// Mitsubishi GX Works2 project: For_daiverter2   PLC: FX3U/FX3UC

PROGRAM MAIN
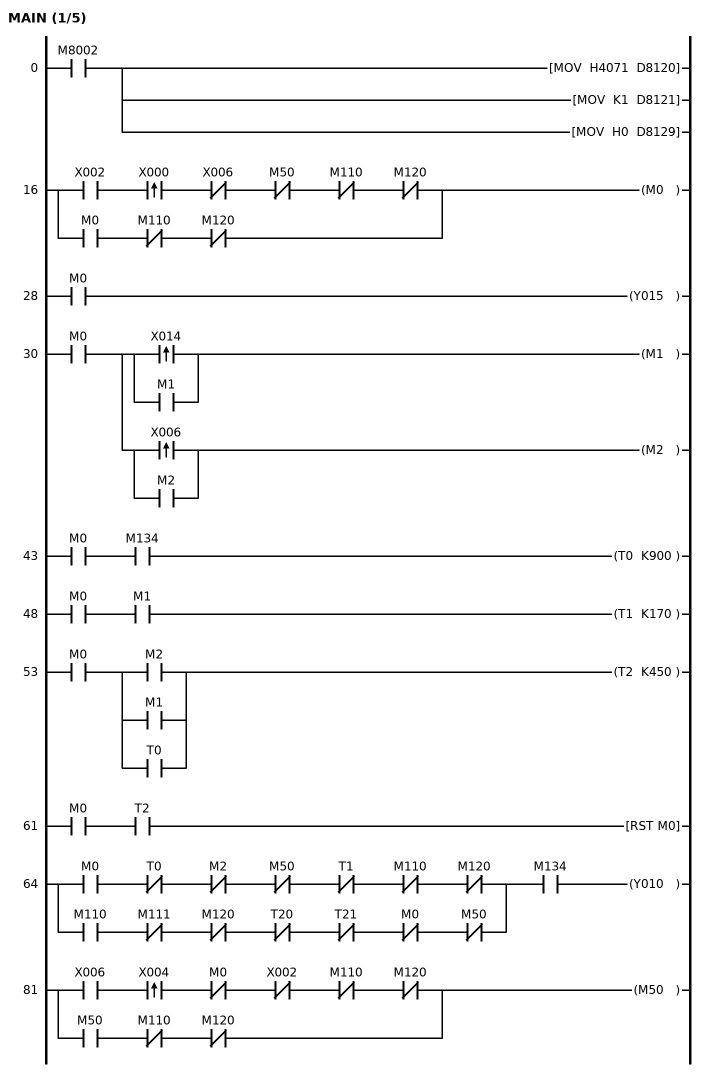
0     LD      M8002
      MOV     H4071 D8120
      MOV     K1 D8121
      MOV     H0 D8129
16    LD      X002
      ANDP    X000
      ANI     X006
      ANI     M50
      ANI     M110
      ANI     M120
      LD      M0
      ANI     M110
      ANI     M120
      ORB
      OUT     M0
28    LD      M0
      OUT     Y015
30    LD      M0
      MPS
      LDP     X014
      OR      M1
      ANB
      OUT     M1
      MPP
      LDP     X006
      OR      M2
      ANB
      OUT     M2
43    LD      M0
      AND     M134
      OUT     T0 K900
48    LD      M0
      AND     M1
      OUT     T1 K170
53    LD      M0
      LD      M2
      OR      M1
      OR      T0
      ANB
      OUT     T2 K450
61    LD      M0
      AND     T2
      RST     M0
64    LD      M0
      ANI     T0
      ANI     M2
      ANI     M50
      ANI     T1
      ANI     M110
      ANI     M120
      LD      M110
      ANI     M111
      ANI     M120
      ANI     T20
      ANI     T21
      ANI     M0
      ANI     M50
      ORB
      AND     M134
      OUT     Y010
81    LD      X006
      ANDP    X004
      ANI     M0
      ANI     X002
      ANI     M110
      ANI     M120
      LD      M50
      ANI     M110
      ANI     M120
      ORB
      OUT     M50
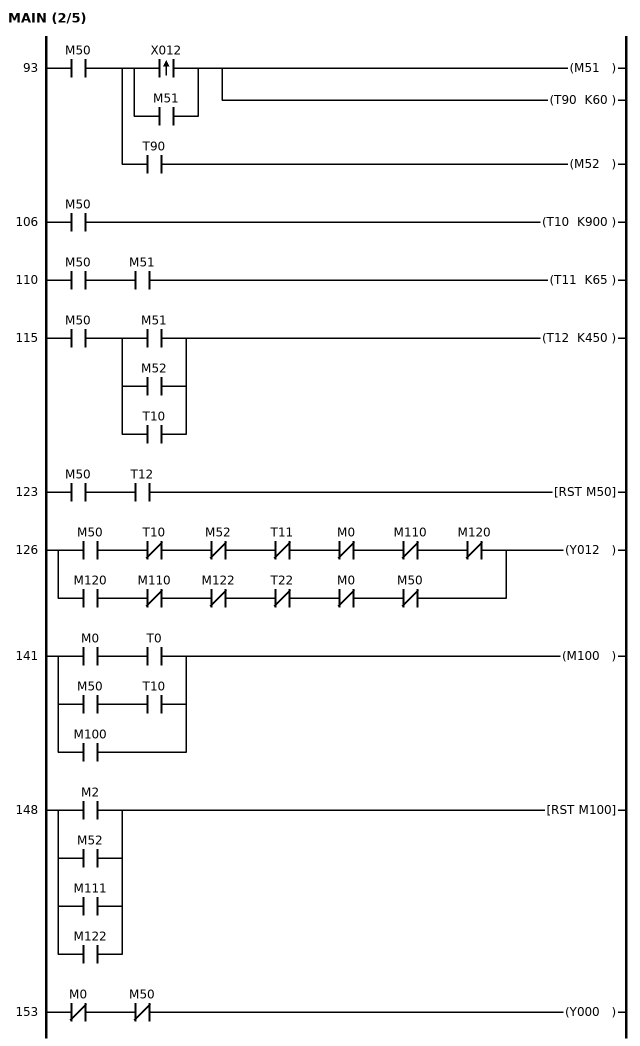
93    LD      M50
      MPS
      LDP     X012
      OR      M51
      ANB
      OUT     M51
      OUT     T90 K60
      MPP
      AND     T90
      OUT     M52
106   LD      M50
      OUT     T10 K900
110   LD      M50
      AND     M51
      OUT     T11 K65
115   LD      M50
      LD      M51
      OR      M52
      OR      T10
      ANB
      OUT     T12 K450
123   LD      M50
      AND     T12
      RST     M50
126   LD      M50
      ANI     T10
      ANI     M52
      ANI     T11
      ANI     M0
      ANI     M110
      ANI     M120
      LD      M120
      ANI     M110
      ANI     M122
      ANI     T22
      ANI     M0
      ANI     M50
      ORB
      OUT     Y012
141   LD      M0
      AND     T0
      LD      M50
      AND     T10
      ORB
      OR      M100
      OUT     M100
148   LD      M2
      OR      M52
      OR      M111
      OR      M122
      RST     M100
153   LDI     M0
      ANI     M50
      OUT     Y000
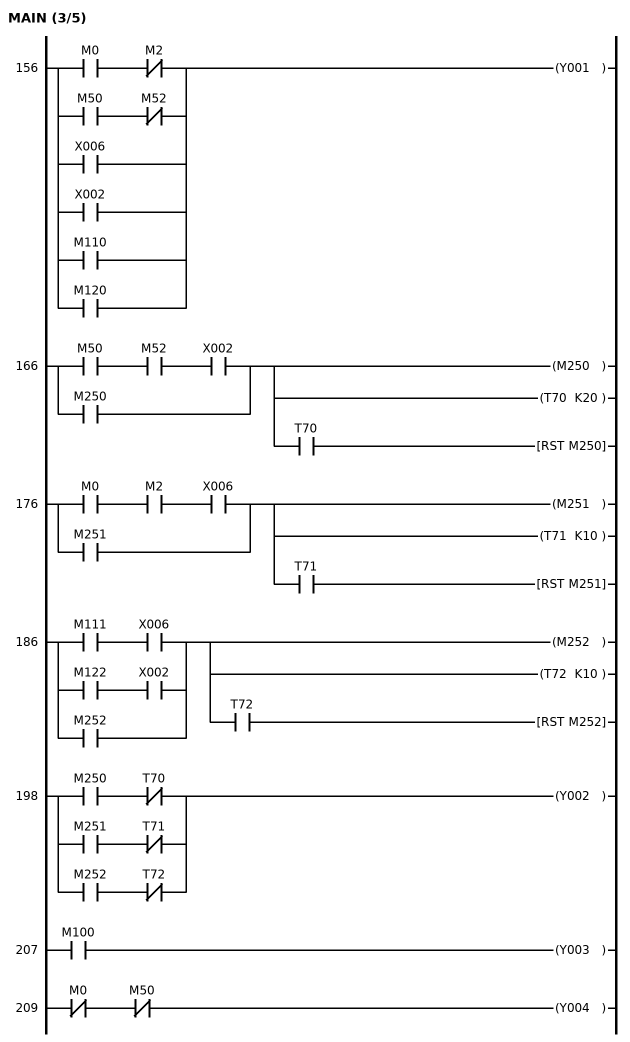
156   LD      M0
      ANI     M2
      LD      M50
      ANI     M52
      ORB
      OR      X006
      OR      X002
      OR      M110
      OR      M120
      OUT     Y001
166   LD      M50
      AND     M52
      AND     X002
      OR      M250
      OUT     M250
      OUT     T70 K20
      AND     T70
      RST     M250
176   LD      M0
      AND     M2
      AND     X006
      OR      M251
      OUT     M251
      OUT     T71 K10
      AND     T71
      RST     M251
186   LD      M111
      AND     X006
      LD      M122
      AND     X002
      ORB
      OR      M252
      OUT     M252
      OUT     T72 K10
      AND     T72
      RST     M252
198   LD      M250
      ANI     T70
      LD      M251
      ANI     T71
      ORB
      LD      M252
      ANI     T72
      ORB
      OUT     Y002
207   LD      M100
      OUT     Y003
209   LDI     M0
      ANI     M50
      OUT     Y004
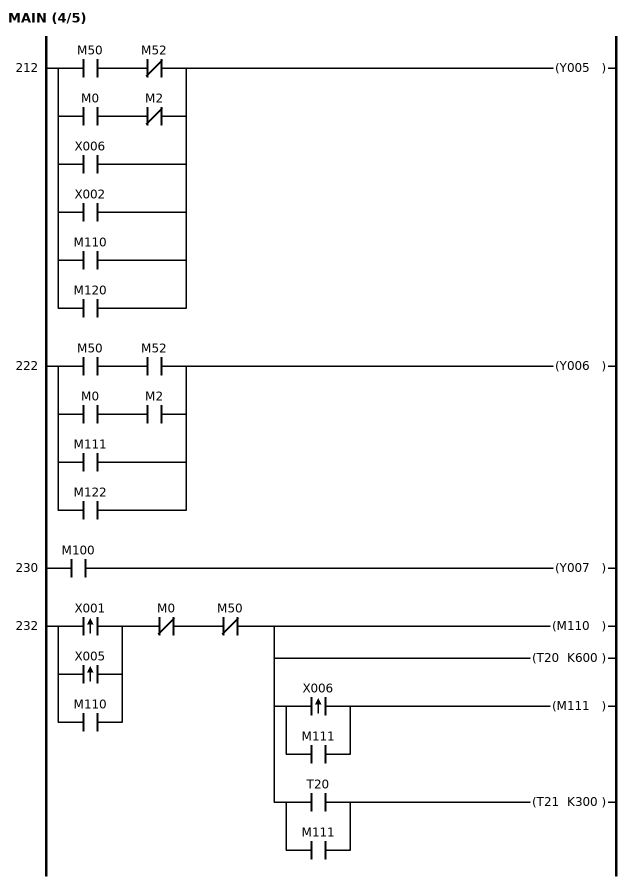
212   LD      M50
      ANI     M52
      LD      M0
      ANI     M2
      ORB
      OR      X006
      OR      X002
      OR      M110
      OR      M120
      OUT     Y005
222   LD      M50
      AND     M52
      LD      M0
      AND     M2
      ORB
      OR      M111
      OR      M122
      OUT     Y006
230   LD      M100
      OUT     Y007
232   LDP     X001
      ORP     X005
      OR      M110
      ANI     M0
      ANI     M50
      OUT     M110
      OUT     T20 K600
      MPS
      LDP     X006
      OR      M111
      ANB
      OUT     M111
      MPP
      LD      T20
      OR      M111
      ANB
      OUT     T21 K300
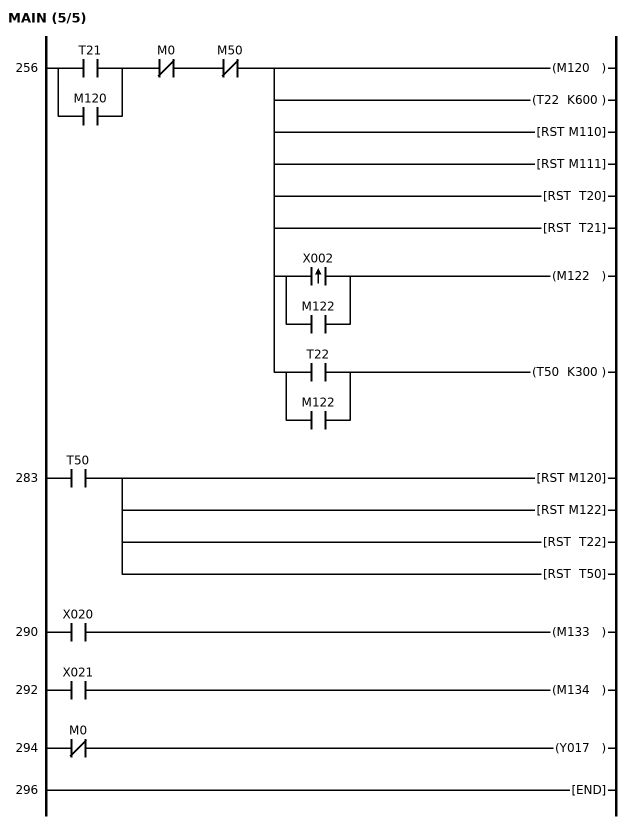
256   LD      T21
      OR      M120
      ANI     M0
      ANI     M50
      OUT     M120
      OUT     T22 K600
      RST     M110
      RST     M111
      RST     T20
      RST     T21
      MPS
      LDP     X002
      OR      M122
      ANB
      OUT     M122
      MPP
      LD      T22
      OR      M122
      ANB
      OUT     T50 K300
283   LD      T50
      RST     M120
      RST     M122
      RST     T22
      RST     T50
290   LD      X020
      OUT     M133
292   LD      X021
      OUT     M134
294   LDI     M0
      OUT     Y017
296   END
END_PROGRAM
